// TIA Portal V20 export
FUNCTION "StepToString" : String   // FC74, SCL
// stored: Namespace Unit1.Em1, SetENOAutomatically false
   VAR_INPUT
      StepDINT : DInt;   // DINT value of the step
   END_VAR
BEGIN
   // Translates the sequence step number to the step name
   // Adjusted for Sequence_1_UnWinder real use case

   CASE #StepDINT OF
       1:
           #StepToString := 'Idle';

       101:
           #StepToString := 'JOB[1] Condition';
       111:
           #StepToString := 'Expel HomePos Check';
       121:
           #StepToString := 'Air Shaft WorkPos Check';
       131:
           #StepToString := 'Radius Measure Check';
       141:
           #StepToString := 'Winder Enable & Control Enable';
       151:
           #StepToString := 'Web Guide EPC Mode Check';
       161:
           #StepToString := 'Tension Sensor Check';
       171:
           #StepToString := 'Bobin ID Check';
       191:
           #StepToString := 'JOB[1] Step End';

       201:
           #StepToString := 'JOB[2] Condition';
       211:
           #StepToString := 'Winder Speed Match Command';
       291:
           #StepToString := 'JOB[2] Step End';

       301:
           #StepToString := 'JOB[3] Condition';
       311:
           #StepToString := 'Winder Speed Match Command';
       391:
           #StepToString := 'JOB[3] Step End';

       401:
           #StepToString := 'JOB[4] Condition';
       411:
           #StepToString := 'Winder Jog BackWard Command';
       421:
           #StepToString := 'Winder Jog BackWard Complete';
       491:
           #StepToString := 'JOB[4] Step End';

       901:
           #StepToString := 'Immediate Stop';

       ELSE
           #StepToString := 'N/A';

   END_CASE;
END_FUNCTION
